FUNCTION_BLOCK RfidHead_Test EXTENDS TcUnit.FB_TestSuite IMPLEMENTS TcoCore.ITcoContext
VAR
    //Context for TcOpen
    _nfContext : TcoCore.TcoContextNfCompatibility;
END_VAR
VAR
    _wrapper_RfidMockNoRfidInRange : RfidMockNoRfidInRange;

    sut_readDataNoTag         : RfidHead(THIS^, _wrapper_RfidMockNoRfidInRange, T#10MS);
    sut_readUidNoTag          : RfidHead(THIS^, _wrapper_RfidMockNoRfidInRange, T#10MS);
    _wrapper_readUid          : RfidMockWorking;
    sut_readUidSuccess        : RfidHead(THIS^, _wrapper_readUid, T#10MS);
    _wrapper_readData         : RfidMockWorking;
    sut_readDataSuccess       : RfidHead(THIS^, _wrapper_readData, T#10MS);
    _wrapper_RfidMockTooLong  : RfidMockWorking;
    sut_readDataTooLongString : RfidHead(THIS^, _wrapper_RfidMockTooLong, T#10MS);
END_VAR

_nfContext.VolatileOpen(); //Required for TCopen
//==============================================

//
//ExecuteReadDataWithTooLongDataLength_ExpectErrorWithErroId();

//
ExecuteReadUidsNoTagInRange_ExpectErrorWithNoTag();
ExecuteReadDataNoTagInRange_ExpectErrorWithNoTag();

//
ExecuteReadUid_ExpectUidAsStringStatusDone();
ExecuteReadData_ExpectDataAsStringStatusDone();

//weitere Tests
// zulange uiDataLength Error
// TimeOut Error
// Lock, Lock mit Error
//==============================================
_nfContext.VolatileClose();

PROPERTY Context : TcoCore.ITcoContext
GET
Context := This^._nfContext;
END_GET
END_PROPERTY

PROPERTY EndCycleCount : ULINT
GET
EndCycleCount := THIS^._nfContext._endCycleCount;
END_GET
END_PROPERTY

PROPERTY Environment : TcoCore.ITcoContextEnvironment
GET
Environment := THIS^._nfContext._settings;
END_GET
END_PROPERTY

METHOD PRIVATE ExecuteReadData_ExpectDataAsStringStatusDone
VAR_INST
    _data          : T_MaxString;
    _expectedData  : T_MaxString := '16# 05 06 07 08';
    _result        : BOOL;
    _udiDataLength : INT := 4;
END_VAR
//{warning disable C0371}
TcUnit.TEST('ExecuteReadData_ExpectDataAsStringStatusDone');
//Arrange
sut_readDataSuccess();

//Act

sut_readDataSuccess.ReadDataMethod(_udiDataLength);
//Assert

IF sut_readDataSuccess.ReadDataTask.Done THEN
    _data := sut_readDataSuccess.Data;

    AssertEquals_STRING(Expected := _expectedData, Actual := _data, Message := 'Daten passt nicht');

    //Busy off
    _result := FALSE;
    AssertEquals_BOOL
    (
        Expected  := _result
        , Actual  := sut_readDataSuccess.ReadDataTask.Busy
        , Message := 'Status Busy muss false sein'
    );

    //Status Done mus True sein
    _result := true;
    AssertEquals_BOOL
    (
        Expected  := _result
        , Actual  := sut_readDataSuccess.ReadDataMethod(_udiDataLength).Done
        , Message := 'Status Done muss true sein'
    );

    //Status Done false again
    sut_readDataSuccess.Restore();
    _result := FALSE;
    AssertEquals_BOOL
    (
        Expected  := _result
        , Actual  := sut_readDataSuccess.ReadDataMethod(_udiDataLength).Done
        , Message := 'Status Done muss false sein nach Reset'
    );

    TcUnit.TEST_FINISHED();
END_IF
END_METHOD

METHOD Private ExecuteReadDataNoTagInRange_ExpectErrorWithNoTag
VAR_INST
    _udiDataLength : INT := 10;
    _result        : BOOL;
    _firstRun      : BOOL := true;
END_VAR
TcUnit.TEST('ExecuteReadDataNoTagInRange_ExpectErrorWithNoTag');

//Assert Initial State
_result := FALSE;

IF _firstRun THEN
    _firstRun := FALSE;
    THIS^.
        AssertEquals_BOOL
    (
        _result
        , sut_readDataNoTag.ReadDataMethod(_udiDataLength).Error
        , 'No Error should be Start Parameter'
    );
END_IF

//Arrange
sut_readDataNoTag();

//Act, Use ReadDataMethod()
sut_readDataNoTag.ReadDataMethod(_udiDataLength);

IF sut_readDataNoTag.ReadDataTask.Error
       OR sut_readUidNoTag.ReadDataTask.Done THEN
    //Assert
    _result := TRUE;

    AssertEquals_BOOL
    (
        _result
        , sut_readDataNoTag.ReadDataMethod(_udiDataLength).Error
        , 'Method did not throw Error'
    );

    AssertEquals_BOOL
    (
        _result
        , sut_readDataNoTag.ReadDataTask.Error
        , 'Task did not throw Error'
    );

    //Act, Restore(), Error shall disappear
    sut_readDataNoTag.Restore();
    _result := FALSE;

    AssertEquals_BOOL
    (
        _result
        , sut_readDataNoTag.ReadDataTask.Error
        , 'Reset did not Work, Still Status Error'
    );

    TcUnit.TEST_FINISHED();
END_IF
END_METHOD

METHOD PRIVATE ExecuteReadDataWithTooLongDataLength_ExpectErrorWithErroId
VAR_INST
    _udiDataLength : INT := 113;
    _result        : BOOL;
    _firstRun      : BOOL := TRUE;

    _errorId : ErrorIDMappingLibraryTurck;

END_VAR
TcUnit.TEST('ExecuteReadDataWithTooLongDataLength_ExpectErrorWithErroId');
//28 blocks, 4 bytes each, => 112 bytes max user Memory!

//Assert Initial State
_result := false;

IF _firstRun THEN
    _firstRun := FALSE;
    THIS^.
        AssertEquals_BOOL
    (
        _result
        , sut_readDataTooLongString.ReadDataMethod(_udiDataLength).Error
        , 'No Error should be Start Parameter'
    );
END_IF

_errorId := sut_readDataTooLongString.ErrorId;

//Arrange
sut_readDataTooLongString();

//Act, Use ReadDataMethod()
sut_readDataTooLongString.ReadDataMethod(_udiDataLength);

IF sut_readDataTooLongString.ReadDataTask.Error
       OR sut_readUidNoTag.ReadDataTask.Done THEN

    _errorId := sut_readDataTooLongString.ErrorId;
    //Assert
    _result := TRUE;

    AssertEquals_BOOL
    (
        _result
        , sut_readDataTooLongString.ReadDataMethod(_udiDataLength).Error
        , 'Method must throw Error'
    );

    AssertEquals_BOOL
    (
        _result
        , sut_readDataTooLongString.ReadDataTask.Error
        , 'Task did not throw Error'
    );

    //Act, Restore(), Error shall disappear
    sut_readDataTooLongString.Restore();
    _result := FALSE;

    AssertEquals_BOOL
    (
        _result
        , sut_readDataTooLongString.ReadDataTask.Error
        , 'Reset did not Work, Still Status Error'
    );

    TcUnit.TEST_FINISHED();
END_IF
END_METHOD

METHOD PRIVATE ExecuteReadUid_ExpectUidAsStringStatusDone
VAR_INST
    _uId         : T_MaxString;
    _expectedUid : T_MaxString := 'E0040150ACF4F3AD';
    _result      : BOOL;
END_VAR
TcUnit.TEST('ExecuteReadUid_ExpectUidAsStringStatusDone');
//Arrange
sut_readUidSuccess();

//Act

sut_readUidSuccess.ReadUidMethod();
//Assert

IF sut_readUidSuccess.ReadUidTask.Done THEN
    _uId := sut_readUidSuccess.Uid;

    AssertEquals_STRING(Expected := _expectedUid, Actual := _uId, Message := 'UID passt nicht');

    //Busy off
    _result := FALSE;
    AssertEquals_BOOL
    (
        Expected  := _result
        , Actual  := sut_readUidSuccess.ReadUidMethod().Busy
        , Message := 'Status Busy muss false sein'
    );

    //Status Done mus True sein
    _result := true;
    AssertEquals_BOOL
    (
        Expected  := _result
        , Actual  := sut_readUidSuccess.ReadUidMethod().Done
        , Message := 'Status Done muss true sein'
    );

    //Status Done false again
    sut_readUidSuccess.Restore();
    _result := FALSE;
    AssertEquals_BOOL
    (
        Expected  := _result
        , Actual  := sut_readUidSuccess.ReadUidMethod().Done
        , Message := 'Status Done muss false sein nach Reset'
    );

    TcUnit.TEST_FINISHED();
END_IF
END_METHOD

METHOD Private ExecuteReadUidsNoTagInRange_ExpectErrorWithNoTag
VAR_INST
    _udiDataLength : INT := 10;
    _result        : BOOL;
    _firstRun      : BOOL := true;
END_VAR
TcUnit.TEST('ExecuteReadUidMethodNoTagInRange_ExpectErrorWithTimeOut');

//Assert Initial State
_result := FALSE;

IF _firstRun THEN
    _firstRun := FALSE;
    THIS^.
        AssertEquals_BOOL
    (
        _result
        , sut_readUidNoTag.ReadDataMethod(_udiDataLength).Error
        , 'No Error should be Start Parameter'
    );
END_IF

//Arrange
sut_readUidNoTag();

//Act, Use ReadUidMethod()
IF sut_readUidNoTag.ReadUidMethod().Error
       OR sut_readUidNoTag.ReadUidMethod().Done THEN
    //Assert
    _result := TRUE;

    AssertEquals_BOOL
    (
        _result
        , sut_readUidNoTag.ReadUidMethod().Error
        , 'Method did not throw Error'
    );

    AssertEquals_BOOL
    (
        _result
        , sut_readUidNoTag.ReadUidTask.Error
        , 'Task did not throw Error'
    );

    //Act, Restore(), Error shall disappear
    sut_readUidNoTag.Restore();
    _result := FALSE;

    AssertEquals_BOOL
    (
        _result
        , sut_readUidNoTag.ReadUidTask.Error
        , 'Reset did not Work, Still Status Error'
    );

    TcUnit.TEST_FINISHED();
END_IF
END_METHOD

PROPERTY Identity : ULINT
GET
Identity := THIS^._nfContext._Identity;
END_GET
END_PROPERTY

PROPERTY Logger : TcoCore.ITcoLogger
GET
Logger := THIS^._nfContext._logger;
END_GET
END_PROPERTY

PROPERTY RealTimeClock : TcoCore.ITcoRtc
GET
RealTimeClock := THIS^._nfContext._rtc;
END_GET
END_PROPERTY

PROPERTY StartCycleCount : ULINT
GET
StartCycleCount := THIS^._nfContext._startCycleCount;
END_GET
END_PROPERTY

END_FUNCTION_BLOCK

(* stored: Version 1.1.0.1, ProductVersion 3.1.4024.12
   POU RfidHead_Test: Id {a47ac61a-ee48-008c-0014-60e0cecfdf35}, SpecialFunc None
   Folder Error: Id {975ec48f-bcf0-0c5d-2b83-0ed4a4227688}
   Folder ITcoContext: Id {33bfe112-ae2f-05c8-0e05-c3229ef70521}
   Folder NoTagError: Id {b5613e50-d453-0eae-3339-03bf860dadda}
   Folder ReadMockWorking: Id {e3a719a8-eedb-0d5a-38a6-6d750e45333d}
   Property Context: Id {7de64d48-d0a2-056e-34b7-aac880c979a6}
   Get Get: Id {9ffe307f-0b04-0675-1acb-4e6595656874}
   Property EndCycleCount: Id {e7bb6f42-b928-0ade-1561-23e4edad0343}
   Get Get: Id {a0db9c75-1b3b-0832-3ccc-1ca1f40db07c}
   Property Environment: Id {e633166a-bd98-0388-2aea-6b9efca83b09}
   Get Get: Id {b02663ba-e6d6-0463-271f-5e82d1a9f4c9}
   Method ExecuteReadData_ExpectDataAsStringStatusDone: Id {7535b2e0-6ab9-065e-2e76-668ef71e8a68}
   Method ExecuteReadDataNoTagInRange_ExpectErrorWithNoTag: Id {ea59a3f7-4d2f-0eda-320a-232679f4280a}
   Method ExecuteReadDataWithTooLongDataLength_ExpectErrorWithErroId: Id {cbc6a826-6270-050b-3244-12340409ff79}
   Method ExecuteReadUid_ExpectUidAsStringStatusDone: Id {4cf9c36f-72dc-08b9-1fac-7b31252a268f}
   Method ExecuteReadUidsNoTagInRange_ExpectErrorWithNoTag: Id {8b561928-65c2-0133-08a7-3dd2d20a1a77}
   Property Identity: Id {1675f325-25d1-008c-3992-a738fcd9949a}
   Get Get: Id {14ac6c95-310e-0e1e-28d6-3f3616785801}
   Property Logger: Id {b14992b0-967b-0e92-3b9d-8efda5b8ea8b}
   Get Get: Id {e7264cb3-b6d7-066e-214a-e06a571621db}
   Property RealTimeClock: Id {150839af-3f34-0d7e-310c-8ded726d6b4f}
   Get Get: Id {26577072-4d1b-0c47-2218-b9aea55e7819}
   Property StartCycleCount: Id {87fd4da8-3313-0074-15f8-03823e1ffcda}
   Get Get: Id {e2f4d863-cdc3-0322-31cb-7a3cd062c769} *)
